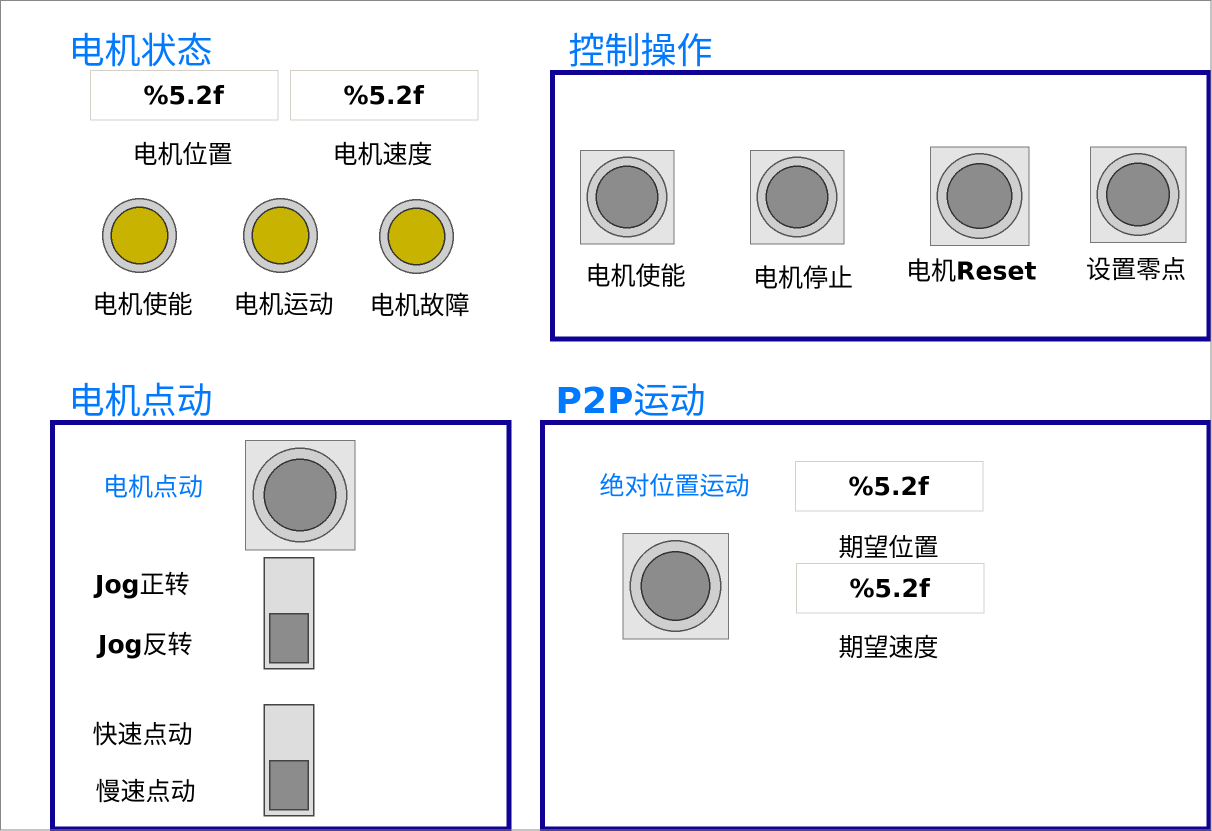
VISUALIZATION Visualization  // 1212x831
    Group (40,20 472x319)
        Group (10,50 462x269)
            Lamp1 (46,120 87x91), variable: Main.motor_state.is_power_ready, style: Lamp-Lamp1-Yellow
            Label (0,200 185x68), "电机使能"
            Textfield (40,0 188x50), "%5.2f", text variable: Main.motor_data.motor_position
            Label (40,50 185x68), "电机位置"
            Textfield (240,0 188x50), "%5.2f", text variable: Main.motor_data.motor_velocity
            Label (240,50 185x68), "电机速度"
            Lamp1 (187,120 87x91), variable: Main.motor_state.is_motor_moving, style: Lamp-Lamp1-Yellow
            Label (141,200 185x68), "电机运动"
            Label (277,201 185x68), "电机故障"
            Lamp1 (323,121 87x91), variable: Main.motor_state.is_motor_error, style: Lamp-Lamp1-Yellow
        Label (0,0 201x61), "电机状态"
    Group (540,20 672x321)
        Rectangle (10,50 661x271)
        Group (20,120 652x165)
            Label (0,110 151x51), "电机使能"
            PushSwitchLed (190,0 94x114), variable: Main.motor_param.is_motor_stop, behaviour: TAP, style: Switch-PushSwitchLed-Gray
            Label (170,110 146x55), "电机停止"
            PushSwitchLed (370,0 99x112), variable: Main.motor_param.is_motor_reset, behaviour: TAP, style: Switch-PushSwitchLed-Gray
            Label (330,110 163x41), "电机Reset"
            PushSwitchLed (530,0 96x109), variable: Main.motor_param.is_set_pos_zero, behaviour: TAP, style: Switch-PushSwitchLed-Gray
            Label (500,110 152x38), "设置零点"
            PushSwitchLed (20,0 94x114), variable: Main.motor_param.is_motor_power_on, behaviour: TAP, style: Switch-PushSwitchLed-Gray
        Label (0,0 201x61), "控制操作"
    Group (40,370 471x461)
        Rectangle (10,50 461x411)
        Group (10,50 310x405)
            Group (0,130 296x128)
                Label (3,60 185x68), "Jog反转"
                DipSwitch (182,7 114x112), variable: Main.motor_param.jog_direction, behaviour: TOGGLE, style: Switch-DipSwitch-Gray
                Label (0,0 185x68), "Jog正转"
            PushSwitchLed (190,20 120x110), variable: Main.motor_param.is_jog_start, behaviour: TAP, style: Switch-PushSwitchLed-Gray
            Label (40,0 126x133), "电机点动"
            Group (0,280 296x125)
                Label (0,0 185x68), "快速点动"
                Label (3,57 185x68), "慢速点动"
                DipSwitch (182,4 114x112), variable: Main.motor_param.jog_mode, behaviour: TOGGLE, style: Switch-DipSwitch-Gray
        Label (0,0 201x61), "电机点动"
    Group (530,370 681x461)
        Rectangle (10,50 671x411)
        Group (20,60 434x251)
            Textfield (245,31 188x50), "%5.2f", text variable: Main.motor_param.move_abs_target_position
                OnMouseClick: write the text variable via Default
            Label (246,83 185x68), "期望位置"
            Label (246,183 185x68), "期望速度"
            Textfield (246,133 188x50), "%5.2f", text variable: Main.motor_param.move_vel
                OnMouseClick: write the text variable via Default
            PushSwitchLed (66,103 119x106), variable: Main.motor_param.is_motor_moving_abs, behaviour: TAP, style: Switch-PushSwitchLed-Gray
            Label (0,0 249x111), "绝对位置运动"
        Label (0,0 201x61), "P2P运动"
END_VISUALIZATION

(* stored: Version 1.1.0.1, ProductVersion 3.1.4024.11
   Visu Visualization: Id {4f144a4b-bbfd-40b9-896b-b5558eeb16b4} *)
